FUNCTION stringCmp : BOOL
VAR_INPUT
	ptStr1 : POINTER TO BYTE;
	ptStr2 : POINTER TO BYTE;
	MaxStringLen	:	UDINT;
END_VAR
VAR
	i				:	UDINT;
END_VAR

StringCmp			:= FALSE;
FOR i := 0 TO MaxStringLen 
DO
   	IF (ptStr1^ <> ptStr2^) 
	THEN  // If two characters are unequal, return FALSE 
      StringCmp 	:= FALSE;
      RETURN;
   	ELSIF ((ptStr1^ = 0) AND (ptStr2^ = 0)) 
	THEN   // If both strings have reached the NULL TERMINATOR at the same place, the strings are identical 
      StringCmp 	:= TRUE;
      RETURN;
   	ELSE						// If the two characters were equal, but were not NULL TERMINATORS, increment to check next character 
      ptStr1 		:= ptStr1 + 1;
      ptStr2 		:= ptStr2 + 1;
   	END_IF
END_FOR

END_FUNCTION

(* stored: Version 1.1.0.1, ProductVersion 3.1.4024.16
   POU stringCmp: Id {594e733b-1b5c-4aae-854c-ba52e0f2610a}, SpecialFunc None *)
